TYPE ENUM_Mirror_State :
(
    Unknown := 0,
    MR1L3In := 1,
    MR1L3Out := 2,
    MR1L3SiC := 3,
    MR1L3W := 4
);
END_TYPE

(* stored: Version 1.1.0.1, ProductVersion 3.1.4022.18
   DUT ENUM_Mirror_State: Id {a0f2074b-5cdf-4540-b535-3ccd590f1f9e} *)
